ABB RobotStudio station: PaletizadoTPL2.rspag

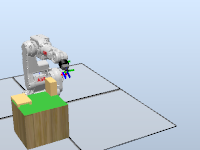
--- station ---
Station Paletizado (saved by RobotStudio 21.1.9443.2)
Controller IRB140_6_81_TPL2
  mechanical unit ROB_1: IRB140_6_81_C_TPL2, 6 joints, base frame (0, 0, 0) mm
Layout (positions relative to the parent item):
  - Mesa [part]
  - Pallet [part]
  - Pieza1 [part]
  - Pieza2 [part]
  - Pieza3 [part]
  - Pieza4 [part]
  - Pieza5 [part]
  - Pieza6 [part]
  - Pieza7 [part]
  - Pieza8 [part] at (0, 0, 0) mm
  - Pieza9 [part] at (0, 0, 0) mm
  - Sopapa [mechanism] at (506.29, 39.79, 679.5) mm, rotated rx 180 ry 60 rz 180 deg
      TCP Sopapa at (0, -5, 103) mm
      links: Sopapa
  - IRB140_6_81_C_TPL2 [mechanism, from Robots\IRB140_6_81_C_G_03.rslib] at (0, 0, 0) mm; joint values [0.0882, 0.0049, -0.0049, -0.1514, 0.5303, 0.175] (rad or m)
Attachment: Sopapa is attached to IRB140_6_81_C_TPL2 / Link6
EventTableEntry 1212: Group=, Trigger=DO_Pinza 1213, Actions=[EventTableActionAttach 1214], Comment=, ActivationMode=2, Cyclic=false
EventTableTriggerIO 1213: IOValue=[1], IRC5Controller=? -1, Operator=0, SignalSource=? -1
EventTableActionAttach 1214: AttachmentParent=Sopapa 1252, AttachmentChild=? -1, MountObject=false, Offset=[X=1, Y=0, Z=0, W=0, X=0, Y=1, Z=0, W=0, X=0, Y=0, Z=1, W=0, X=0, Y=0, Z=0, W=1], FlangeIndext=0, FindNearest=true
EventTableEntry 1219: Group=, Trigger=DO_Pinza 1220, Actions=[EventTableActionDetach 1221], Comment=, ActivationMode=2, Cyclic=false
EventTableTriggerIO 1220: IOValue=[0], IRC5Controller=? -1, Operator=0, SignalSource=? -1
EventTableActionDetach 1221: AttachmentParent=Sopapa 1252, AttachmentChild=? -1

--- Backups/IRB140_6_81_TPL2/RAPID/TASK1/PROGMOD/Module1.mod ---
MODULE Module1
    PERS tooldata Sopapa:=[TRUE,[[0,-5,103],[1,0,0,0]],[.500,[0,0,40],[1,0,0,0],0,0,0]];
    CONST robtarget Target_10:=[[595.492267836,-5,628],[0.5,0,0.866025404,0],[0,0,0,0],[9E+09,9E+09,9E+09,9E+09,9E+09,9E+09]];
    CONST robtarget Target_20:=[[595.492192643,34.78927249,628.000011052],[0.500000018,0.000000003,0.866025394,0.000000005],[0,-1,0,0],[9E+09,9E+09,9E+09,9E+09,9E+09,9E+09]];
!***********************************************************
    !
    ! Module:  Module1
    !
    ! Description:
    !   <Insert description here>
    !
    ! Author: CARTELLI
    !
    ! Version: 1.0
    !
    !***********************************************************


    !***********************************************************
    !
    ! Procedure main
    !
    !   This is the entry point of your program
    !
    !***********************************************************
    PROC main()
        !Add your code here
        Path_10;
    ENDPROC
    PROC Path_10()
        MoveL Target_10,v1000,z100,Sopapa\WObj:=wobj0;
        MoveL Target_20,v1000,z100,Sopapa\WObj:=wobj0;
    ENDPROC
ENDMODULE
